// TIA Portal V16 export
// export: Created 2024-09-05T17:40:14.9767109Z, ExportSetting WithDefaults, DisplayName Totally Integrated Automation Portal, DisplayVersion V16 Update 6, DisplayName TIA Portal Version Control Interface, DisplayVersion V16 Update 2, DisplayName TIA Portal Openness, DisplayVersion V16 Update 6, DisplayName STEP 7 Professional, DisplayVersion V16 Update 6, DisplayName STEP 7 Safety, DisplayVersion V16, DisplayName WinCC Advanced, DisplayVersion V16 Update 6
TYPE "UDT_Results_Cupforming"
// stored: IsFailsafeCompliant false
   STRUCT
      MaxForce : Real;
      MinimalWay : Real;
      MaxZposition : Real;
      OK : Bool;
      NOK : Bool;
      parameters : "UDT_FittingParameters";
   END_STRUCT;
END_TYPE
